KUKA KRL data list: wkz4_ab.dat

&ACCESS RVO9
&REL 231
&COMMENT Deposita Pinca C3
&PARAM DISKPATH = KRC:\R1\Program
DEFDAT  wkz4_ab
;FOLD EXTERNAL DECLARATIONS;%{PE}%MKUKATPBASIS,%CEXT,%VCOMMON,%P
;FOLD GRIPPERTECH EXT
EXT  H50 (INT  :IN,INT  :IN,INT  :IN,GRP_TYP  :IN )
;ENDFOLD (GRIPPERTECH EXT)
;FOLD SPOTTECH EXT
EXT  USERSPOT (S_COMMAND  :IN,SPOT_TYPE  :IN )
;ENDFOLD (SPOTTECH EXT)
;FOLD BASISTECH EXT;%{PE}%MKUKATPBASIS,%CEXT,%VEXT,%P
EXT  BAS (BAS_COMMAND  :IN,REAL  :IN )
DECL INT SUCCESS
;ENDFOLD (BASISTECH EXT)
;FOLD USER EXT;%{E}%MKUKATPUSER,%CEXT,%VEXT,%P
;Make your modifications here

;ENDFOLD (USER EXT)
;ENDFOLD (EXTERNAL DECLARATIONS)

;# ============ START PATH : zh_p13060r2_c1 =============
DECL E6POS XLHP015={X -308.16391,Y -965.055725,Z 1491.62097,A 110.519302,B -4.6375699,C 90.9493866,S 18,T 2,E1 0.0,E2 0.0,E3 0.0,E4 0.0,E5 0.0,E6 0.0}
DECL FDAT FLHP015={TOOL_NO 4,BASE_NO 0,IPO_FRAME #BASE,TQ_STATE FALSE}
DECL PDAT PPDAT21={VEL 100.0,ACC 93.0,APO_DIST 65.0,APO_MODE #CDIS}
DECL E6POS XLHP025={X -1221.08496,Y -1499.32898,Z 1268.12598,A 127.241699,B -0.116557099,C 90.6040192,S 18,T 2,E1 0.0,E2 0.0,E3 0.0,E4 0.0,E5 0.0,E6 0.0}
DECL FDAT FLHP025={TOOL_NO 4,BASE_NO 0,IPO_FRAME #BASE,TQ_STATE FALSE}
DECL E6POS XPDEPOSITO={X -1306.89502,Y -1563.30005,Z 577.696899,A 136.741302,B -0.541404486,C 89.859993,S 18,T 2,E1 0.0,E2 0.0,E3 0.0,E4 0.0,E5 0.0,E6 0.0}
DECL FDAT FpDeposito={TOOL_NO 4,BASE_NO 0,IPO_FRAME #BASE,TQ_STATE FALSE}
DECL E6POS XLHP035={X -936.369812,Y -915.347717,Z 957.483215,A 151.736206,B -0.176963001,C 179.617798,S 18,T 2,E1 0.0,E2 0.0,E3 0.0,E4 0.0,E5 0.0,E6 0.0}
DECL FDAT FLHP035={TOOL_NO 8,BASE_NO 0,IPO_FRAME #BASE,TQ_STATE FALSE}
DECL LDAT LCPDAT14={VEL 2.0,ACC 100.0,APO_DIST 100.0,APO_FAC 50.0}
DECL E6POS XLHP030={X -1239.19202,Y -1602.31995,Z 904.860229,A 136.518097,B -0.465419114,C 89.911087,S 18,T 2,E1 0.0,E2 0.0,E3 0.0,E4 0.0,E5 0.0,E6 0.0}
DECL FDAT FLHP030={TOOL_NO 4,BASE_NO 0,IPO_FRAME #BASE,TQ_STATE FALSE}
DECL E6POS XLHP045={X -222.850098,Y -954.188477,Z 1457.18298,A 161.598007,B 1.35442996,C -174.552094,S 18,T 10,E1 0.0,E2 0.0,E3 0.0,E4 0.0,E5 0.0,E6 0.0}
DECL FDAT FLHP045={TOOL_NO 8,BASE_NO 0,IPO_FRAME #BASE,TQ_STATE FALSE}
DECL PDAT PPDAT34={VEL 100.0,ACC 100.0,APO_DIST 100.0,APO_MODE #CDIS}
DECL E6POS XLHP040={X -936.471313,Y -915.518921,Z 1183.34998,A 151.735397,B -0.178353205,C 179.602402,S 18,T 2,E1 0.0,E2 0.0,E3 0.0,E4 0.0,E5 0.0,E6 0.0}
DECL FDAT FLHP040={TOOL_NO 8,BASE_NO 0,IPO_FRAME #BASE,TQ_STATE FALSE}
DECL PDAT PPDAT35={VEL 100.0,ACC 100.0,APO_DIST 100.0,APO_MODE #CDIS}
DECL E6POS XLHP010={X 274.967407,Y -867.433411,Z 1505.20605,A 140.761902,B -4.28091002,C 91.8909836,S 18,T 34,E1 0.0,E2 0.0,E3 0.0,E4 0.0,E5 0.0,E6 0.0}
DECL FDAT FLHP010={TOOL_NO 4,BASE_NO 0,IPO_FRAME #BASE,TQ_STATE FALSE}
DECL PDAT PPDAT36={VEL 100.0,ACC 100.0,APO_DIST 20.0,APO_MODE #CDIS}
DECL GRP_SUGG_T LAST_GRP={NUMBER[] "1                       ",STATE[] "1                       ",PARAMS[] "GDAT0                   "}
DECL SPOT_SUGG_T LAST_SPOT={GUN[] "1                       ",RETR_CMD[] "#OPN                    ",CHOISE[] "#FIRST                  ",CLO_TM[] "1                       ",PGNO1[] "1                       ",PRESS1[] "0                       ",PGNO2[] "1                       ",PRESS2[] "0                       ",SPOT_PARAMS[] "NORMAL                  "}
DECL BASIS_SUGG_T LAST_BASIS={POINT1[] "P0                      ",POINT2[] "P0                      ",CP_PARAMS[] "CPDAT0                  ",PTP_PARAMS[] "PDAT0                   ",CONT[] "                        ",CP_VEL[] "2.0                     ",PTP_VEL[] " 100                    ",SYNC_PARAMS[] "SYNCDAT                 ",SPL_NAME[] "S0                      "}
DECL PDAT PPDAT1={VEL 100.0,ACC 100.0,APO_DIST 10.0,APO_MODE #CDIS,GEAR_JERK 50.0}
DECL E6POS XLHP016={X -898.836609,Y -1025.16797,Z 1464.76794,A 108.922501,B -1.28892696,C 89.1518021,S 18,T 2,E1 0.0,E2 0.0,E3 0.0,E4 0.0,E5 0.0,E6 0.0}
DECL FDAT FLHP016={TOOL_NO 4,BASE_NO 0,IPO_FRAME #BASE,POINT2[] " ",TQ_STATE FALSE}
DECL PDAT PPDAT2={VEL 100.0,ACC 100.0,APO_DIST 100.0,APO_MODE #CDIS,GEAR_JERK 50.0}
DECL PDAT PPDAT4={VEL 100.0,ACC 93.0,APO_DIST 65.0,APO_MODE #CDIS,GEAR_JERK 50.0}
DECL E6POS XLHP031={X -1307.36499,Y -1561.21899,Z 757.031372,A 136.741394,B -0.5467152,C 89.8438568,S 18,T 2,E1 0.0,E2 0.0,E3 0.0,E4 0.0,E5 0.0,E6 0.0}
DECL FDAT FLHP031={TOOL_NO 4,BASE_NO 0,IPO_FRAME #BASE,POINT2[] " ",TQ_STATE FALSE}
DECL LDAT LCPDAT1={VEL 2.0,ACC 100.0,APO_DIST 100.0,APO_FAC 50.0,AXIS_VEL 100.0,AXIS_ACC 100.0,ORI_TYP #VAR,CIRC_TYP #BASE,JERK_FAC 50.0,GEAR_JERK 50.0,EXAX_IGN 0}
DECL E6POS XLHP050={X 493.744995,Y -685.626709,Z 1450.30396,A -173.494705,B 6.03480816,C -171.047897,S 18,T 10,E1 0.0,E2 0.0,E3 0.0,E4 0.0,E5 0.0,E6 0.0}
DECL FDAT FLHP050={TOOL_NO 8,BASE_NO 0,IPO_FRAME #BASE,POINT2[] " ",TQ_STATE FALSE}
DECL PDAT PPDAT6={VEL 100.0,ACC 100.0,APO_DIST 100.0,APO_MODE #CDIS,GEAR_JERK 50.0}
DECL E6POS XLHP055={X 1015.54901,Y 298.872101,Z 1632.73804,A -38.790081,B -12.1412096,C -163.671097,S 18,T 3,E1 0.0,E2 0.0,E3 0.0,E4 0.0,E5 0.0,E6 0.0}

DECL FDAT FLHP055={TOOL_NO 8,BASE_NO 0,IPO_FRAME #BASE,POINT2[] " ",TQ_STATE FALSE}
DECL PDAT PPDAT7={VEL 100.0,ACC 100.0,APO_DIST 100.0,APO_MODE #CDIS,GEAR_JERK 50.0}
DECL LDAT LCPDAT3={VEL 2.0,ACC 100.0,APO_DIST 100.0,APO_FAC 50.0,AXIS_VEL 100.0,AXIS_ACC 100.0,ORI_TYP #VAR,CIRC_TYP #BASE,JERK_FAC 50.0,GEAR_JERK 50.0,EXAX_IGN 0}
DECL E6POS XP2={X 22.4985104,Y 1240.30896,Z 1237.56201,A -46.9696198,B 1.22592998,C 179.895203,S 18,T 11,E1 0.0,E2 0.0,E3 0.0,E4 0.0,E5 0.0,E6 0.0}
DECL FDAT FP2={TOOL_NO 8,BASE_NO 0,IPO_FRAME #BASE,POINT2[] " ",TQ_STATE FALSE}
DECL PDAT PPDAT11={VEL 100.0,ACC 100.0,APO_DIST 100.0,APO_MODE #CDIS,GEAR_JERK 50.0}
DECL E6POS XP3={X 859.804382,Y 543.648987,Z 1516.61694,A -110.137199,B -3.30189395,C 90.8716431,S 18,T 3,E1 0.0,E2 0.0,E3 0.0,E4 0.0,E5 0.0,E6 0.0}
DECL FDAT FP3={TOOL_NO 4,BASE_NO 0,IPO_FRAME #BASE,POINT2[] " ",TQ_STATE FALSE}
DECL PDAT PPDAT12={VEL 100.0,ACC 100.0,APO_DIST 20.0,APO_MODE #CDIS,GEAR_JERK 50.0}
DECL E6POS XP4={X -1307.36597,Y -1561.15601,Z 679.818481,A 136.740601,B -0.545101285,C 89.8497314,S 18,T 2,E1 0.0,E2 0.0,E3 0.0,E4 0.0,E5 0.0,E6 0.0}
DECL FDAT FP4={TOOL_NO 4,BASE_NO 0,IPO_FRAME #BASE,POINT2[] " ",TQ_STATE FALSE}
DECL LDAT LCPDAT5={VEL 2.0,ACC 100.0,APO_DIST 100.0,APO_FAC 50.0,AXIS_VEL 100.0,AXIS_ACC 100.0,ORI_TYP #VAR,CIRC_TYP #BASE,JERK_FAC 50.0,GEAR_JERK 50.0,EXAX_IGN 0}
DECL E6POS XP5={X 248.530899,Y 1766.22998,Z 1797.63,A -10.4337702,B 3.25291395,C 113.526497,S 18,T 11,E1 0.0,E2 0.0,E3 0.0,E4 0.0,E5 0.0,E6 0.0}
DECL FDAT FP5={TOOL_NO 4,BASE_NO 0,IPO_FRAME #BASE,POINT2[] " ",TQ_STATE FALSE}
DECL PDAT PPDAT20={VEL 100.0,ACC 100.0,APO_DIST 100.0,GEAR_JERK 50.0}
DECL PDAT PPDAT22={VEL 50.0,ACC 100.0,APO_DIST 100.0,GEAR_JERK 50.0}
DECL E6POS XSWP_60_0401={X 4359.27881,Y -4196.02881,Z -267.779388,A -135.832794,B -1.47759199,C 89.4332428,S 18,T 2,E1 0.0,E2 0.0,E3 0.0,E4 0.0,E5 0.0,E6 0.0}
DECL FDAT FSWP_60_0401={TOOL_NO 4,BASE_NO 2,IPO_FRAME #BASE,POINT2[] " "}
DECL PDAT PPDAT23={VEL 100.0,ACC 100.0,APO_DIST 100.0,APO_MODE #CDIS,GEAR_JERK 50.0}
DECL E6POS XP6={X -848.207214,Y -960.370789,Z 1217.11096,A 149.435593,B -0.121127501,C 179.868195,S 18,T 2,E1 0.0,E2 0.0,E3 0.0,E4 0.0,E5 0.0,E6 0.0}
DECL FDAT FP6={TOOL_NO 8,BASE_NO 0,IPO_FRAME #BASE,POINT2[] " ",TQ_STATE FALSE}
DECL E6POS XP1={X 799.621277,Y 800.155823,Z 1739.07898,A -96.5585403,B 4.41296387,C 88.0835571,S 18,T 11,E1 0.0,E2 0.0,E3 0.0,E4 0.0,E5 0.0,E6 0.0}
DECL FDAT FP1={TOOL_NO 4,BASE_NO 0,IPO_FRAME #BASE,POINT2[] " ",TQ_STATE FALSE}
DECL PDAT PPDAT3={VEL 100.0,ACC 100.0,APO_DIST 100.0,APO_MODE #CDIS,GEAR_JERK 50.0}
ENDDAT
